// TIA Portal project "FactoryIO_Template_S7-1200_V15_V15.1_V18" (V18)
// Vorlageprojekt für das Buch mit Zielsystem S7-1200

(* hardware
DEVICE "S7-1200-Station_1"  S7-1200 Station
   slot 0: "Baugruppenträger_0"  Rack  V1.0
   slot 1: "PLC_1"  CPU 1214FC DC/DC/RLY  6ES7 214-1HF40-0XB0  V4.6
   slot 2: "DI 16/DQ 16x24VDC_1"  6ES7 223-1BL32-0XB0  V2.0
   slot 3: "DQ 16x24VDC_1"  SM 1222 DQ16 x 24VDC  6ES7 222-1BH32-0XB0  V2.0
   slot 3: "DQ 4x24VDC_1"  DQ4 signal board (200 kHz)  6ES7 222-1BD30-0XB0  V1.0
   slot 4: "DQ 16x24VDC_2"  SM 1222 DQ16 x 24VDC  6ES7 222-1BH32-0XB0  V2.0
   slot 5: "DQ 16x24VDC_3"  SM 1222 DQ16 x 24VDC  6ES7 222-1BH32-0XB0  V2.0
*)

// ===== PLC "PLC_1"  CPU 1214FC DC/DC/RLY =====

VAR_GLOBAL   // PLC tag table "Standard-Variablentabelle"
   "At Entry" AT %I5.0 : Bool;
   "At Load" AT %I5.1 : Bool;
   "At Left" AT %I5.2 : Bool;
   "At Middle" AT %I5.3 : Bool;
   "At Right" AT %I5.4 : Bool;
   "At Unload" AT %I5.5 : Bool;
   "At Exit" AT %I5.6 : Bool;
   "Moving X" AT %I5.7 : Bool;
   "Moving Z" AT %I6.0 : Bool;
   "Старт" AT %I6.1 : Bool;
   "Стоп" AT %I6.2 : Bool;
   "Сброс счетчика (ячейки)" AT %I6.3 : Bool;
   "Завоз на склад" AT %I6.4 : Bool;
   "Вывоз со склада" AT %I6.5 : Bool;
   "Entry Conveyor" AT %Q10.0 : Bool;
   "Load Conveyor" AT %Q10.1 : Bool;
   "Forks Left" AT %Q10.2 : Bool;
   "Forks Right" AT %Q10.3 : Bool;
   "Lift" AT %Q10.4 : Bool;
   "Unload Conveyor" AT %Q10.5 : Bool;
   "Exit Conveyor" AT %Q10.6 : Bool;
   "Старт (лампа)" AT %Q10.7 : Bool;
   "Стоп (лампа)" AT %Q11.0 : Bool;
   "Завозящие конвейеры" AT %M0.0 : Bool;
   "Вывозящие конвейеры" AT %M0.6 : Bool;
   "Перемещение предмета" AT %M0.1 : Bool;
   "Движение по какой-то из осей" AT %M0.2 : Bool;
   "Вернулся с грузом" AT %M0.4 : Bool;
   "Возврат лифта" AT %M0.3 : Bool;
   "Ячейка убрана" AT %M0.5 : Bool;
   "Ячейка" AT %QD12 : DInt;
   "По правую сторону" AT %M0.7 : Bool;
   "Вывод занятых ячеек" AT %QD16 : Real;
END_VAR

// folder: System blocks/Program resources

DATA_BLOCK "IEC_Timer_0_DB_8"   // DB10
{ S7_Optimized_Access := 'TRUE' }
AUTHOR : Simatic
FAMILY : IEC
NAME : IEC_TMR
VERSION : 1.0
// stored: InstanceOfName IEC_TIMER
"IEC_TIMER"
BEGIN
END_DATA_BLOCK

DATA_BLOCK "IEC_Timer_0_DB_9"   // DB11
{ S7_Optimized_Access := 'TRUE' }
AUTHOR : Simatic
FAMILY : IEC
NAME : IEC_TMR
VERSION : 1.0
// stored: InstanceOfName IEC_TIMER
"IEC_TIMER"
BEGIN
END_DATA_BLOCK

DATA_BLOCK "IEC_Timer_0_DB_10"   // DB12
{ S7_Optimized_Access := 'TRUE' }
AUTHOR : Simatic
FAMILY : IEC
NAME : IEC_TMR
VERSION : 1.0
// stored: InstanceOfName IEC_TIMER
"IEC_TIMER"
BEGIN
END_DATA_BLOCK

DATA_BLOCK "IEC_Timer_0_DB_11"   // DB13
{ S7_Optimized_Access := 'TRUE' }
AUTHOR : Simatic
FAMILY : IEC
NAME : IEC_TMR
VERSION : 1.0
// stored: InstanceOfName IEC_TIMER
"IEC_TIMER"
BEGIN
END_DATA_BLOCK

DATA_BLOCK "IEC_Counter_0_DB_1"   // DB14
{ S7_Optimized_Access := 'TRUE' }
AUTHOR : SIMATIC
FAMILY : IEC
NAME : DCNTR
VERSION : 1.2
// stored: InstanceOfName IEC_DCOUNTER
"IEC_DCOUNTER"
BEGIN
END_DATA_BLOCK

DATA_BLOCK "IEC_Timer_0_DB_12"   // DB15
{ S7_Optimized_Access := 'TRUE' }
AUTHOR : Simatic
FAMILY : IEC
NAME : IEC_TMR
VERSION : 1.0
// stored: InstanceOfName IEC_TIMER
"IEC_TIMER"
BEGIN
END_DATA_BLOCK

DATA_BLOCK "IEC_Timer_0_DB_13"   // DB16
{ S7_Optimized_Access := 'TRUE' }
AUTHOR : Simatic
FAMILY : IEC
NAME : IEC_TMR
VERSION : 1.0
// stored: InstanceOfName IEC_TIMER
"IEC_TIMER"
BEGIN
END_DATA_BLOCK

// folder: (top level)

FUNCTION "MHJ-PLC-Lab-Function-S71200" : Void   // FC9000, SCL
{ S7_Optimized_Access := 'TRUE' }
VERSION : 0.1
   VAR_TEMP
      rdTimeReturn : Int;
      outputTime : DTL;
      SyncVal : Byte;
      forVal : Int;
      forVal_2 : Int;
      Value : Byte;
   END_VAR
   VAR CONSTANT
      CompVal : Byte := 16#34;
      Value_01 : Byte := 16#11;
      Value_01_DW : DWord := 16#A165_D992;
      Value_02_DW : DWord := 16#58BE_4401;
   END_VAR
BEGIN

   #Value:=PEEK(area := 16#82,
        dbNumber := 0,
        byteOffset := 511);
   #Value := #Value + 1;

   POKE(area := 16#82,
        dbNumber := 0,
        byteOffset := 511,
        value := #Value);

   POKE(area:=16#81,
        dbNumber:=0,
        byteOffset:=1016,
        value:=#Value_01_DW);
   POKE(area := 16#81,
        dbNumber := 0,
        byteOffset := 1020,
        value := #Value_02_DW);

   POKE(area := 16#81,
        dbNumber := 0,
        byteOffset := 511,
        value := B#16#00);

   FOR #forVal := 0 TO 120 DO
       FOR #forVal_2:=0 TO 10 DO
           #rdTimeReturn:=RD_SYS_T(#outputTime);
           #rdTimeReturn := WR_SYS_T(#outputTime);
           #rdTimeReturn := RD_SYS_T(#outputTime);
           #rdTimeReturn := WR_SYS_T(#outputTime);
       END_FOR;
       #SyncVal:= PEEK(area := 16#81,
                      dbNumber := 0,
                      byteOffset := 511);
       IF #SyncVal = #CompVal THEN
          GOTO M_1;
       END_IF;
   END_FOR;
   RETURN;

   M_1:
   POKE(area := 16#81,
        dbNumber := 0,
        byteOffset := 511,
        value := B#16#0);
END_FUNCTION

ORGANIZATION_BLOCK "Main"   // OB1, LAD, ProgramCycle
TITLE = "Main Program Sweep (Cycle)"
{ S7_Optimized_Access := 'TRUE' }
VERSION : 0.1
// ППч
   VAR_INPUT
      Initial_Call : Bool;   // Initial call of this OB
      Remanence : Bool;   // =True, if remanent data are available
   END_VAR
   VAR_TEMP   // added for the SCL form of the ladder/FBD networks
      _w1 : Bool;
      _w2 : Bool;
      _w3 : Bool;
      _w4 : Bool;
      _w5 : Bool;
      _w6 : Bool;
      _w7 : Bool;
      _w8 : Bool;
   END_VAR
BEGIN

REGION Network 1: Konnektierungsbaustein für PLC-Lab / Связь с Factory IO
   // Im Netzwerk 1 wird der Konnektierungsbaustein für PLC-Lab aufgerufen.
   // Dieser Aufruf darf nicht entfernt werden!
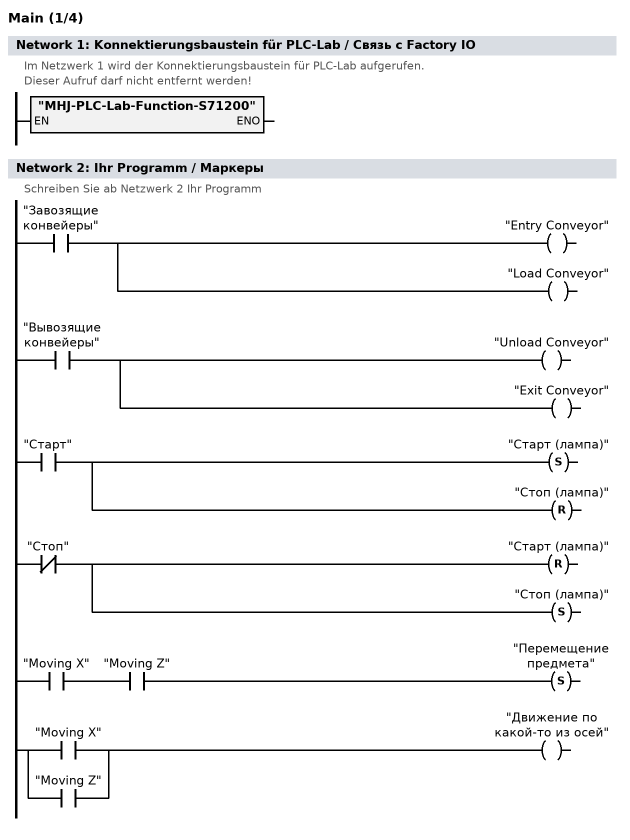
   RUNG wire#powerrail
      "MHJ-PLC-Lab-Function-S71200"()
   END_RUNG
   // the same network as SCL:
   "MHJ-PLC-Lab-Function-S71200"();
END_REGION

REGION Network 2: Ihr Programm / Маркеры
   // Schreiben Sie ab Netzwerk 2 Ihr Programm
   RUNG wire#powerrail
      Contact( "Завозящие конвейеры" )
      wire#w1
      Coil( "Entry Conveyor" )
   END_RUNG
   RUNG wire#w1
      Coil( "Load Conveyor" )
   END_RUNG
   RUNG wire#powerrail
      Contact( "Вывозящие конвейеры" )
      wire#w2
      Coil( "Unload Conveyor" )
   END_RUNG
   RUNG wire#w2
      Coil( "Exit Conveyor" )
   END_RUNG
   RUNG wire#powerrail
      Contact( "Старт" )
      wire#w3
      S_Coil( "Старт (лампа)" )
   END_RUNG
   RUNG wire#w3
      R_Coil( "Стоп (лампа)" )
   END_RUNG
   RUNG wire#powerrail
      I_Contact( "Стоп" )
      wire#w4
      R_Coil( "Старт (лампа)" )
   END_RUNG
   RUNG wire#w4
      S_Coil( "Стоп (лампа)" )
   END_RUNG
   RUNG wire#powerrail
      Contact( "Moving X" )
      Contact( "Moving Z" )
      S_Coil( "Перемещение предмета" )
   END_RUNG
   RUNG wire#powerrail
      Contact( "Moving X" )
      wire#w5
      Coil( "Движение по какой-то из осей" )
   END_RUNG
   RUNG wire#powerrail
      Contact( "Moving Z" )
   END_RUNG wire#w5
   // the same network as SCL:
   "Entry Conveyor" := "Завозящие конвейеры";
   "Load Conveyor" := "Завозящие конвейеры";
   "Unload Conveyor" := "Вывозящие конвейеры";
   "Exit Conveyor" := "Вывозящие конвейеры";
   IF "Старт" THEN
       "Старт (лампа)" := TRUE;
       "Стоп (лампа)" := FALSE;
   END_IF;
   IF NOT "Стоп" THEN
       "Старт (лампа)" := FALSE;
       "Стоп (лампа)" := TRUE;
   END_IF;
   IF "Moving X" AND "Moving Z" THEN "Перемещение предмета" := TRUE; END_IF;
   "Движение по какой-то из осей" := "Moving X" OR "Moving Z";
END_REGION

REGION Network 3: Завоз к складу
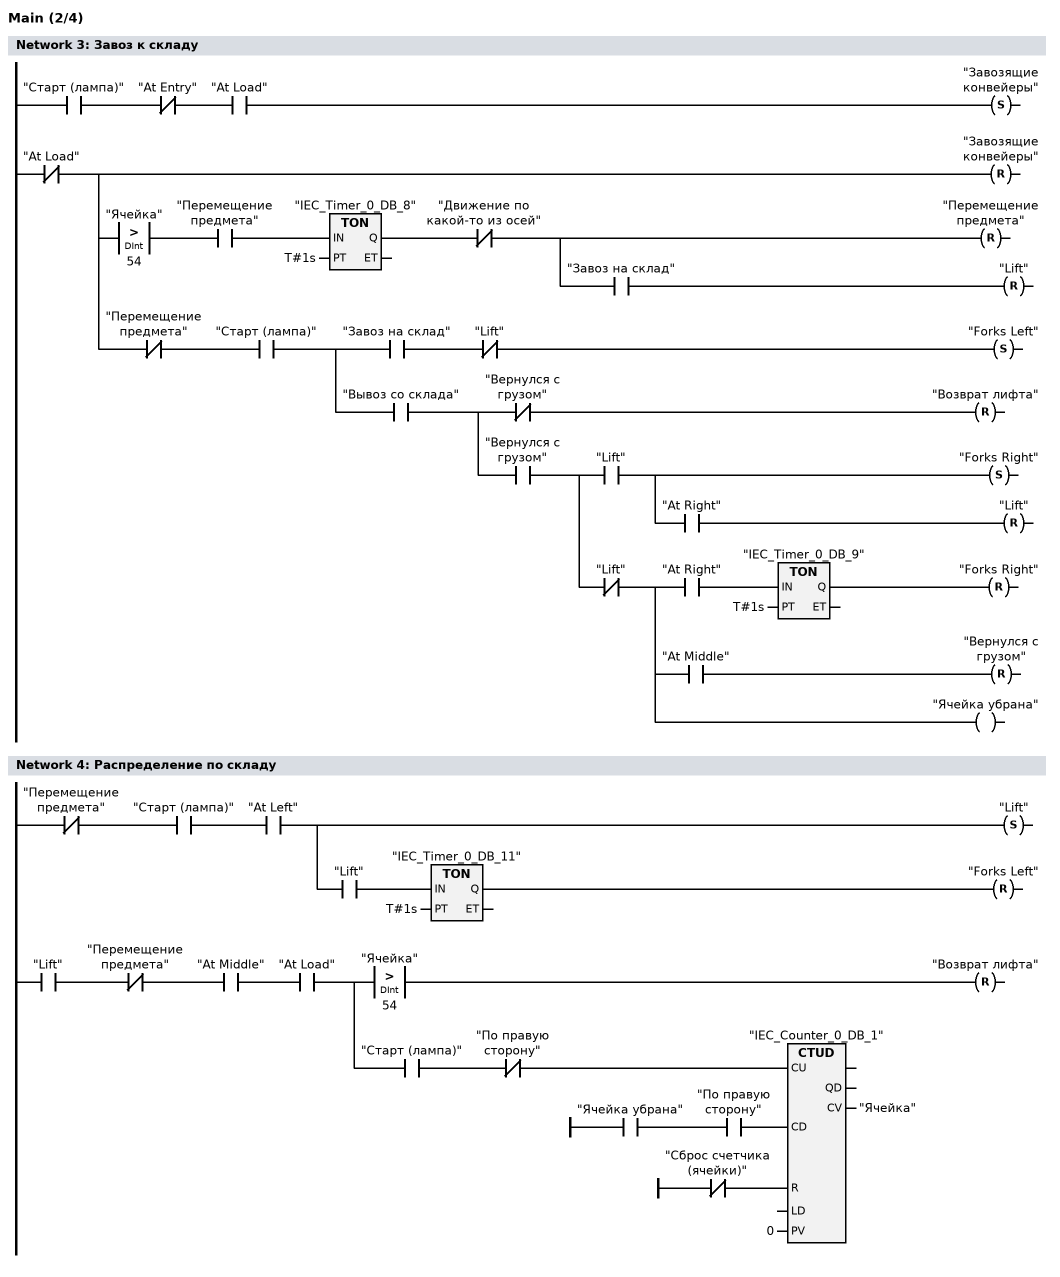
   IF "Старт (лампа)" AND NOT "At Entry" AND "At Load" THEN "Завозящие конвейеры" := TRUE; END_IF;
   IF NOT "At Load" THEN "Завозящие конвейеры" := FALSE; END_IF;
   "IEC_Timer_0_DB_8".TON(IN := NOT "At Load" AND ("Ячейка" > 54) AND "Перемещение предмета", PT := T#1s);
   #_w1 := "IEC_Timer_0_DB_8".Q AND NOT "Движение по какой-то из осей";
   IF #_w1 THEN "Перемещение предмета" := FALSE; END_IF;
   IF #_w1 AND "Завоз на склад" THEN "Lift" := FALSE; END_IF;
   #_w2 := NOT "At Load" AND NOT "Перемещение предмета" AND "Старт (лампа)";
   IF #_w2 AND "Завоз на склад" AND NOT "Lift" THEN "Forks Left" := TRUE; END_IF;
   #_w3 := #_w2 AND "Вывоз со склада";
   IF #_w3 AND NOT "Вернулся с грузом" THEN "Возврат лифта" := FALSE; END_IF;
   #_w4 := #_w3 AND "Вернулся с грузом";
   #_w5 := #_w4 AND "Lift";
   IF #_w5 THEN "Forks Right" := TRUE; END_IF;
   IF #_w5 AND "At Right" THEN "Lift" := FALSE; END_IF;
   #_w6 := #_w4 AND NOT "Lift";
   "IEC_Timer_0_DB_9".TON(IN := #_w6 AND "At Right", PT := T#1s);
   IF "IEC_Timer_0_DB_9".Q THEN "Forks Right" := FALSE; END_IF;
   IF #_w6 AND "At Middle" THEN "Вернулся с грузом" := FALSE; END_IF;
   "Ячейка убрана" := #_w6;
END_REGION

REGION Network 4: Распределение по складу
   #_w1 := NOT "Перемещение предмета" AND "Старт (лампа)" AND "At Left";
   IF #_w1 THEN "Lift" := TRUE; END_IF;
   "IEC_Timer_0_DB_11".TON(IN := #_w1 AND "Lift", PT := T#1s);
   IF "IEC_Timer_0_DB_11".Q THEN "Forks Left" := FALSE; END_IF;
   #_w2 := "Lift" AND NOT "Перемещение предмета" AND "At Middle" AND "At Load";
   IF #_w2 AND ("Ячейка" > 54) THEN "Возврат лифта" := FALSE; END_IF;
   "IEC_Counter_0_DB_1".CTUD(CU := #_w2 AND "Старт (лампа)" AND NOT "По правую сторону",
                           CD := "Ячейка убрана" AND "По правую сторону",
                           R := NOT "Сброс счетчика (ячейки)",
                           PV := 0,
                           CV => "Ячейка");
END_REGION

REGION Network 5: Возврат лифта и действия на стеллаже
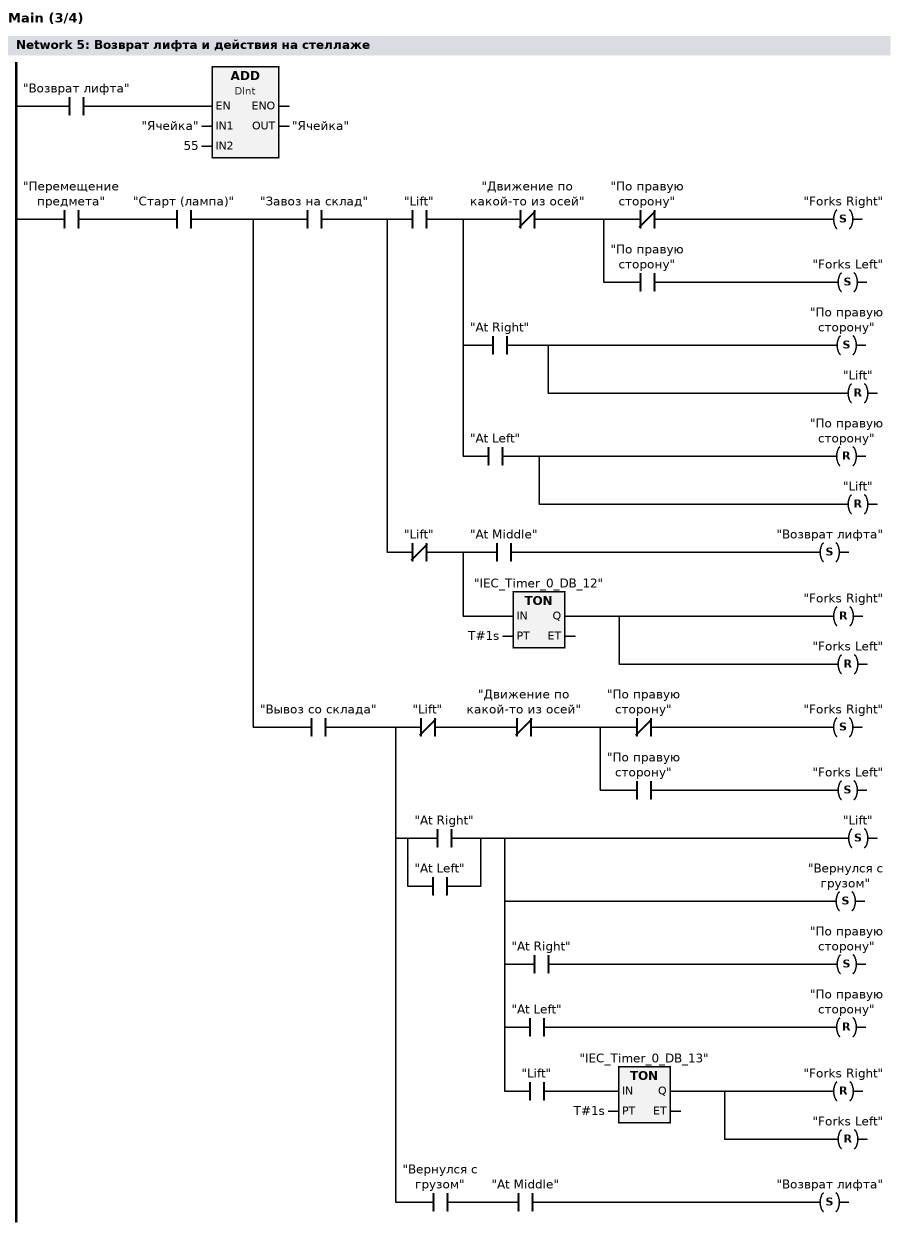
   IF "Возврат лифта" THEN "Ячейка" := "Ячейка" + 55; END_IF;
   #_w1 := "Перемещение предмета" AND "Старт (лампа)";
   #_w2 := #_w1 AND "Завоз на склад";
   #_w3 := #_w2 AND "Lift";
   #_w4 := #_w3 AND NOT "Движение по какой-то из осей";
   IF #_w4 AND NOT "По правую сторону" THEN "Forks Right" := TRUE; END_IF;
   IF #_w4 AND "По правую сторону" THEN "Forks Left" := TRUE; END_IF;
   IF #_w3 AND "At Right" THEN
       "По правую сторону" := TRUE;
       "Lift" := FALSE;
   END_IF;
   IF #_w3 AND "At Left" THEN
       "По правую сторону" := FALSE;
       "Lift" := FALSE;
   END_IF;
   #_w5 := #_w2 AND NOT "Lift";
   IF #_w5 AND "At Middle" THEN "Возврат лифта" := TRUE; END_IF;
   "IEC_Timer_0_DB_12".TON(IN := #_w5, PT := T#1s);
   IF "IEC_Timer_0_DB_12".Q THEN
       "Forks Right" := FALSE;
       "Forks Left" := FALSE;
   END_IF;
   #_w6 := #_w1 AND "Вывоз со склада";
   #_w7 := #_w6 AND NOT "Lift" AND NOT "Движение по какой-то из осей";
   IF #_w7 AND NOT "По правую сторону" THEN "Forks Right" := TRUE; END_IF;
   IF #_w7 AND "По правую сторону" THEN "Forks Left" := TRUE; END_IF;
   #_w8 := #_w6 AND ("At Right" OR "At Left");
   IF #_w8 THEN
       "Lift" := TRUE;
       "Вернулся с грузом" := TRUE;
   END_IF;
   IF #_w8 AND "At Right" THEN "По правую сторону" := TRUE; END_IF;
   IF #_w8 AND "At Left" THEN "По правую сторону" := FALSE; END_IF;
   "IEC_Timer_0_DB_13".TON(IN := #_w8 AND "Lift", PT := T#1s);
   IF "IEC_Timer_0_DB_13".Q THEN
       "Forks Right" := FALSE;
       "Forks Left" := FALSE;
   END_IF;
   IF #_w6 AND "Вернулся с грузом" AND "At Middle" THEN "Возврат лифта" := TRUE; END_IF;
END_REGION

REGION Network 6: Вывоз со склада
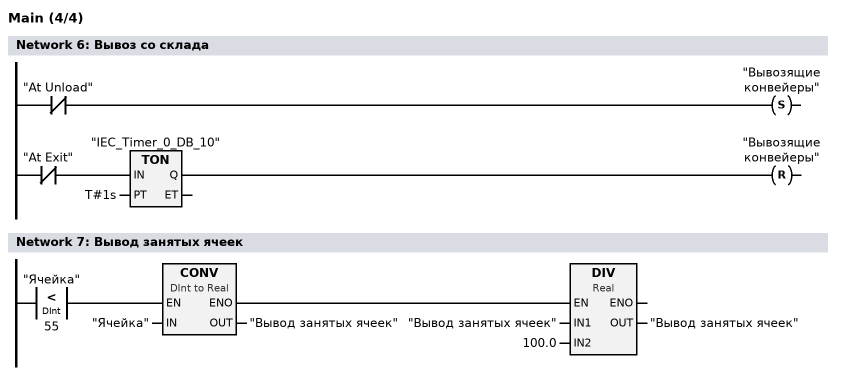
   IF NOT "At Unload" THEN "Вывозящие конвейеры" := TRUE; END_IF;
   "IEC_Timer_0_DB_10".TON(IN := NOT "At Exit", PT := T#1s);
   IF "IEC_Timer_0_DB_10".Q THEN "Вывозящие конвейеры" := FALSE; END_IF;
END_REGION

REGION Network 7: Вывод занятых ячеек
   RUNG wire#powerrail
      { S7_Templates := "SrcType := DInt" } LT_Contact(in1 := "Ячейка", in2 := 55)
      { S7_Templates := "[SrcType := DInt, DestType := Real]" } Convert(in := "Ячейка", out => "Вывод занятых ячеек")
      { S7_Templates := "SrcType := Real" } Div(in1 := "Вывод занятых ячеек", in2 := 100.0, out => "Вывод занятых ячеек")
   END_RUNG
   // the same network as SCL:
   IF "Ячейка" < 55 THEN
       "Вывод занятых ячеек" := DINT_TO_REAL("Ячейка");
       "Вывод занятых ячеек" := "Вывод занятых ячеек" / 100.0;
   END_IF;
END_REGION
END_ORGANIZATION_BLOCK